TYPE E_OriType :
(
	eOT_Var := 0,
	eOT_Constant,
	eOT_Joint
);
END_TYPE

(* stored: Version 1.1.0.1, ProductVersion 3.1.4020.12
   DUT E_OriType: Id {63bf06af-42cd-480b-a437-5b9c1b4c32e1} *)
